PROGRAM POURunLight
VAR
END_VAR

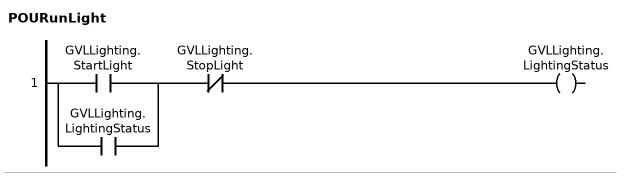
// NETWORK 1
GVLLighting.LightingStatus := (GVLLighting.StartLight OR GVLLighting.LightingStatus) AND NOT GVLLighting.StopLight;

END_PROGRAM

(* stored: Version 1.1.0.1, ProductVersion 3.1.4022.3
   POU POURunLight: Id {7e6ea83a-f1ad-4a4b-a2d7-af6a915eeb93}, SpecialFunc None *)
